(* IEC 61131-3 sources: AXOpen/src/components.cognex.vision/ctrl/test, 5 files *)

(* ---- AxoDatamanTests.st ---- *)
USING AXOpen.Core;
USING AXOpen.Messaging;
USING AXOpen.Messaging.Static;

// Tests for AxoDataman (Cognex Dataman v6.0.0 code reader).
//
// AxoDataman.Run(inParent, hwID) performs PROFINET hardware-slot introspection
// (ReadSlotFromHardwareID / ReadHardwareIDFromSlot / ReadHardwareIOAddress) before any
// inspection logic. On the LLVM unit-test simulator there is no real PROFINET device, so
// the "settled inspection" happy path is not reachable here (it requires real hardware).
// What IS deterministic on the simulator is the input-guard / hardware-resolution error
// path: those branches set a fixed Status.Error.Id and are exercised below. Expected IDs
// are the component's own documented guard constants (TROUBLES.md is a stub).
NAMESPACE Cognex.Vision.Tests.Dataman
    {S7.extern=ReadWrite}
    CLASS TestContext EXTENDS AXOpen.Core.Dummies.MockAxoContext
        METHOD PROTECTED OVERRIDE Main
            ;
        END_METHOD
    END_CLASS

    {TestFixture}
    {S7.extern=ReadWrite}
    CLASS AxoDatamanTests
        VAR
            context : TestContext;
            sut     : AXOpen.Components.Cognex.Vision.v_6_0_0_0.AxoDataman;
            parent  : AXOpen.Core.AxoObject;
            _rtc    : AXOpen.Core.Dummies.MockAxoRtc;
            _rtm    : AXOpen.Core.Dummies.MockAxoRtm;
            _nullParent : IAxoObject;   // unassigned interface reference == NULL
        END_VAR

        VAR
            contextBlank : TestContext;
            sutBlank     : AXOpen.Components.Cognex.Vision.v_6_0_0_0.AxoDataman;
            parentBlank  : AXOpen.Core.AxoObject;
        END_VAR

        {TestSetup}
        METHOD PUBLIC TestSetup
            context := contextBlank;
            sut     := sutBlank;
            parent  := parentBlank;
            _rtm.SetElapsed(LTIME#2s);
            context.InjectRtm(_rtm);
            _rtc.SetNowUTC(LDATE_AND_TIME#2012-01-12-15:58:12.123);
            context.InjectRtc(_rtc);
            context.InitializeRootObject(parent);
        END_METHOD

        // inParent == NULL is a programming error -> Status.Error.Id := 700.
        {Test}
        METHOD PUBLIC Run_WithNullParent_RaisesError700
            context.Open();
            sut.Run(_nullParent, UINT#16);
            context.Close();

            AxUnit.Assert.Equal(UINT#700, sut.Status.Error.Id);
        END_METHOD

        // hwID == 0 (no device hardware identifier) is a programming error -> 701.
        {Test}
        METHOD PUBLIC Run_WithZeroHardwareId_RaisesError701
            context.Open();
            context.InitializeRootObject(parent);
            sut.Run(parent, UINT#0);
            context.Close();

            AxUnit.Assert.Equal(UINT#701, sut.Status.Error.Id);
        END_METHOD

        // A non-zero hwID resolves the device, but slot 1 (AcquisitionControl) cannot be
        // resolved on the simulator (the unmocked hardware reads return default 0) -> 710.
        {Test}
        METHOD PUBLIC Run_WithoutHardwarePresent_RaisesSlotError710
            context.Open();
            context.InitializeRootObject(parent);
            sut.Run(parent, UINT#16);
            context.Close();

            AxUnit.Assert.Equal(UINT#710, sut.Status.Error.Id);
        END_METHOD
    END_CLASS
END_NAMESPACE

(* ---- AxoInsightV24Tests.st ---- *)
USING AXOpen.Core;
USING AXOpen.Messaging;
USING AXOpen.Messaging.Static;

// Tests for AxoInsight v24.0.0 (Cognex In-Sight 2800 vision sensor).
//
// As with the v6 variant, Run(inParent, hwID) performs PROFINET hardware-slot introspection
// before any vision logic, so on the LLVM simulator only the input-guard / hardware-resolution
// error path is deterministically reachable. Expected IDs are the component's guard constants.
NAMESPACE Cognex.Vision.Tests.InsightV24
    {S7.extern=ReadWrite}
    CLASS TestContext EXTENDS AXOpen.Core.Dummies.MockAxoContext
        METHOD PROTECTED OVERRIDE Main
            ;
        END_METHOD
    END_CLASS

    {TestFixture}
    {S7.extern=ReadWrite}
    CLASS AxoInsightV24Tests
        VAR
            context : TestContext;
            sut     : AXOpen.Components.Cognex.Vision.v_24_0_0.AxoInsight;
            parent  : AXOpen.Core.AxoObject;
            _rtc    : AXOpen.Core.Dummies.MockAxoRtc;
            _rtm    : AXOpen.Core.Dummies.MockAxoRtm;
            _nullParent : IAxoObject;
        END_VAR

        VAR
            contextBlank : TestContext;
            sutBlank     : AXOpen.Components.Cognex.Vision.v_24_0_0.AxoInsight;
            parentBlank  : AXOpen.Core.AxoObject;
        END_VAR

        {TestSetup}
        METHOD PUBLIC TestSetup
            context := contextBlank;
            sut     := sutBlank;
            parent  := parentBlank;
            _rtm.SetElapsed(LTIME#2s);
            context.InjectRtm(_rtm);
            _rtc.SetNowUTC(LDATE_AND_TIME#2012-01-12-15:58:12.123);
            context.InjectRtc(_rtc);
            context.InitializeRootObject(parent);
        END_METHOD

        {Test}
        METHOD PUBLIC Run_WithNullParent_RaisesError700
            context.Open();
            sut.Run(_nullParent, UINT#16);
            context.Close();

            AxUnit.Assert.Equal(UINT#700, sut.Status.Error.Id);
        END_METHOD

        {Test}
        METHOD PUBLIC Run_WithZeroHardwareId_RaisesError701
            context.Open();
            context.InitializeRootObject(parent);
            sut.Run(parent, UINT#0);
            context.Close();

            AxUnit.Assert.Equal(UINT#701, sut.Status.Error.Id);
        END_METHOD

        {Test}
        METHOD PUBLIC Run_WithoutHardwarePresent_RaisesSlotError710
            context.Open();
            context.InitializeRootObject(parent);
            sut.Run(parent, UINT#16);
            context.Close();

            AxUnit.Assert.Equal(UINT#710, sut.Status.Error.Id);
        END_METHOD
    END_CLASS
END_NAMESPACE

(* ---- AxoInsightV6Tests.st ---- *)
USING AXOpen.Core;
USING AXOpen.Messaging;
USING AXOpen.Messaging.Static;

// Tests for AxoInsight v6.0.0 (Cognex In-Sight vision sensor).
//
// AxoInsight.Run(inParent, hwID) performs PROFINET hardware-slot introspection before any
// vision logic. On the LLVM unit-test simulator there is no real PROFINET device, so the
// settled inspection happy path is not reachable here. The deterministic, simulator-runnable
// behaviour is the input-guard / hardware-resolution error path; expected IDs are the
// component's own guard constants.
NAMESPACE Cognex.Vision.Tests.InsightV6
    {S7.extern=ReadWrite}
    CLASS TestContext EXTENDS AXOpen.Core.Dummies.MockAxoContext
        METHOD PROTECTED OVERRIDE Main
            ;
        END_METHOD
    END_CLASS

    {TestFixture}
    {S7.extern=ReadWrite}
    CLASS AxoInsightV6Tests
        VAR
            context : TestContext;
            sut     : AXOpen.Components.Cognex.Vision.v_6_0_0_0.AxoInsight;
            parent  : AXOpen.Core.AxoObject;
            _rtc    : AXOpen.Core.Dummies.MockAxoRtc;
            _rtm    : AXOpen.Core.Dummies.MockAxoRtm;
            _nullParent : IAxoObject;
        END_VAR

        VAR
            contextBlank : TestContext;
            sutBlank     : AXOpen.Components.Cognex.Vision.v_6_0_0_0.AxoInsight;
            parentBlank  : AXOpen.Core.AxoObject;
        END_VAR

        {TestSetup}
        METHOD PUBLIC TestSetup
            context := contextBlank;
            sut     := sutBlank;
            parent  := parentBlank;
            _rtm.SetElapsed(LTIME#2s);
            context.InjectRtm(_rtm);
            _rtc.SetNowUTC(LDATE_AND_TIME#2012-01-12-15:58:12.123);
            context.InjectRtc(_rtc);
            context.InitializeRootObject(parent);
        END_METHOD

        {Test}
        METHOD PUBLIC Run_WithNullParent_RaisesError700
            context.Open();
            sut.Run(_nullParent, UINT#16);
            context.Close();

            AxUnit.Assert.Equal(UINT#700, sut.Status.Error.Id);
        END_METHOD

        {Test}
        METHOD PUBLIC Run_WithZeroHardwareId_RaisesError701
            context.Open();
            context.InitializeRootObject(parent);
            sut.Run(parent, UINT#0);
            context.Close();

            AxUnit.Assert.Equal(UINT#701, sut.Status.Error.Id);
        END_METHOD

        {Test}
        METHOD PUBLIC Run_WithoutHardwarePresent_RaisesSlotError710
            context.Open();
            context.InitializeRootObject(parent);
            sut.Run(parent, UINT#16);
            context.Close();

            AxUnit.Assert.Equal(UINT#710, sut.Status.Error.Id);
        END_METHOD
    END_CLASS
END_NAMESPACE

(* ---- AxoVisionProNetTests.st ---- *)
USING AXOpen.Core;
USING AXOpen.Messaging;
USING AXOpen.Messaging.Static;

// Tests for AxoVisionProNet (Cognex VisionPro over a TCP/.NET remote-task channel).
//
// Unlike the PROFINET variants, Run(inParent) performs NO hardware-slot introspection, so the
// component runs end-to-end on the LLVM simulator. Its data-exchange tasks are AxoRemoteTasks
// whose handlers live on the .NET twin, which is not present under `apax test`; therefore these
// tests cover only twin-independent, deterministic behaviour:
//   * a clean cyclic Run leaves the component error-free (Status.ErrorCode = 0),
//   * Restore() clears Status (ErrorCode/Accepted/descriptions) per the docs,
//   * manual control gates the commissioning task (IsManuallyControllable after activation).
// Remote-task busy/done/exception states (which depend on the missing twin handler) are not
// asserted.
NAMESPACE Cognex.Vision.Tests.VisionProNet
    {S7.extern=ReadWrite}
    CLASS TestContext EXTENDS AXOpen.Core.Dummies.MockAxoContext
        METHOD PROTECTED OVERRIDE Main
            ;
        END_METHOD
    END_CLASS

    {TestFixture}
    {S7.extern=ReadWrite}
    CLASS AxoVisionProNetTests
        VAR
            context : TestContext;
            sut     : AXOpen.Components.Cognex.Vision.AxoVisionProNet;
            parent  : AXOpen.Core.AxoObject;
            _rtc    : AXOpen.Core.Dummies.MockAxoRtc;
            _rtm    : AXOpen.Core.Dummies.MockAxoRtm;
        END_VAR

        VAR
            contextBlank : TestContext;
            sutBlank     : AXOpen.Components.Cognex.Vision.AxoVisionProNet;
            parentBlank  : AXOpen.Core.AxoObject;
        END_VAR

        {TestSetup}
        METHOD PUBLIC TestSetup
            context := contextBlank;
            sut     := sutBlank;
            parent  := parentBlank;
            _rtm.SetElapsed(LTIME#2s);
            context.InjectRtm(_rtm);
            _rtc.SetNowUTC(LDATE_AND_TIME#2012-01-12-15:58:12.123);
            context.InjectRtc(_rtc);
            context.InitializeRootObject(parent);
        END_METHOD

        METHOD PRIVATE Cycle
            context.Open();
            context.InitializeRootObject(parent);
            sut.Run(parent);
            context.Close();
        END_METHOD

        // A clean cyclic run with nothing invoked leaves the component free of error.
        {Test}
        METHOD PUBLIC Run_WhenIdle_KeepsErrorCodeZero
            VAR i : INT; END_VAR
            FOR i := 0 TO 3 DO
                THIS.Cycle();
            END_FOR;

            AxUnit.Assert.Equal(INT#0, sut.Status.ErrorCode);
        END_METHOD

        // Restore() clears the status fields back to their initial state.
        {Test}
        METHOD PUBLIC Restore_ClearsStatus
            THIS.Cycle();

            // dirty the status, then restore
            sut.Status.ErrorCode := INT#42;
            sut.Status.Accepted  := TRUE;

            context.Open();
            context.InitializeRootObject(parent);
            sut.Restore();
            sut.Run(parent);
            context.Close();

            AxUnit.Assert.Equal(INT#0, sut.Status.ErrorCode);
            AxUnit.Assert.Equal(FALSE, sut.Status.Accepted);
        END_METHOD

        // After ActivateManualControl(), the component reports itself manually controllable
        // for the activating context cycle (and the next), per AxoComponent semantics.
        {Test}
        METHOD PUBLIC ManualControl_WhenActivated_IsManuallyControllable
            THIS.Cycle();              // bind the component to the context

            sut.ActivateManualControl();
            THIS.Cycle();              // evaluate manual-control state within the window

            AxUnit.Assert.Equal(TRUE, sut.IsManuallyControllable());
        END_METHOD
    END_CLASS
END_NAMESPACE

(* ---- AxoVisionProTests.st ---- *)
USING AXOpen.Core;
USING AXOpen.Messaging;
USING AXOpen.Messaging.Static;

// Tests for AxoVisionPro (Cognex VisionPro over PROFINET, multi-camera).
//
// Run(inParent, hwID, CameraNo) performs extensive PROFINET hardware-slot introspection
// (17 slots) before any vision logic. On the LLVM simulator there is no real PROFINET device,
// so the settled inspection happy path is not reachable here. The deterministic,
// simulator-runnable behaviour is the input-guard / hardware-resolution error path; expected
// IDs are the component's guard constants.
NAMESPACE Cognex.Vision.Tests.VisionPro
    {S7.extern=ReadWrite}
    CLASS TestContext EXTENDS AXOpen.Core.Dummies.MockAxoContext
        METHOD PROTECTED OVERRIDE Main
            ;
        END_METHOD
    END_CLASS

    {TestFixture}
    {S7.extern=ReadWrite}
    CLASS AxoVisionProTests
        VAR
            context : TestContext;
            sut     : AXOpen.Components.Cognex.Vision.AxoVisionPro;
            parent  : AXOpen.Core.AxoObject;
            _rtc    : AXOpen.Core.Dummies.MockAxoRtc;
            _rtm    : AXOpen.Core.Dummies.MockAxoRtm;
            _nullParent : IAxoObject;
        END_VAR

        VAR
            contextBlank : TestContext;
            sutBlank     : AXOpen.Components.Cognex.Vision.AxoVisionPro;
            parentBlank  : AXOpen.Core.AxoObject;
        END_VAR

        {TestSetup}
        METHOD PUBLIC TestSetup
            context := contextBlank;
            sut     := sutBlank;
            parent  := parentBlank;
            _rtm.SetElapsed(LTIME#2s);
            context.InjectRtm(_rtm);
            _rtc.SetNowUTC(LDATE_AND_TIME#2012-01-12-15:58:12.123);
            context.InjectRtc(_rtc);
            context.InitializeRootObject(parent);
        END_METHOD

        {Test}
        METHOD PUBLIC Run_WithNullParent_RaisesError700
            context.Open();
            sut.Run(_nullParent, UINT#16, BYTE#1);
            context.Close();

            AxUnit.Assert.Equal(UINT#700, sut.Status.Error.Id);
        END_METHOD

        {Test}
        METHOD PUBLIC Run_WithZeroHardwareId_RaisesError701
            context.Open();
            context.InitializeRootObject(parent);
            sut.Run(parent, UINT#0, BYTE#1);
            context.Close();

            AxUnit.Assert.Equal(UINT#701, sut.Status.Error.Id);
        END_METHOD

        // Non-zero hwID resolves the device, but slot 1 (SystemControl) cannot be resolved on
        // the simulator (unmocked hardware reads return default 0) -> 710.
        {Test}
        METHOD PUBLIC Run_WithoutHardwarePresent_RaisesSlotError710
            context.Open();
            context.InitializeRootObject(parent);
            sut.Run(parent, UINT#16, BYTE#1);
            context.Close();

            AxUnit.Assert.Equal(UINT#710, sut.Status.Error.Id);
        END_METHOD
    END_CLASS
END_NAMESPACE
